Yaskawa INFORM job: R1_W35-36-A2(90,0)KM-OK_MOD.JBI

/JOB
//NAME R1_W35-36-A2(90,0)KM-OK_MOD
///FOLDERNAME KRIS-SCIANA
//POS
///NPOS 134,134,0,9,0,0
///TOOL 0
///POSTYPE PULSE
///PULSE
C00000=-14538,91541,13322,-12188,94395,86333
C00001=-53862,-64636,-102244,-12188,94395,-55972
C00002=-133203,-148839,-120155,9781,61912,-66404
C00003=-174797,-117438,-114286,21839,44085,-72130
C00004=-167772,-84651,-94857,14466,47220,-68129
C00005=-165686,-79015,-89435,12794,46452,-67294
C00006=-164380,-75470,-85062,11842,45407,-66832
C00007=-163956,-74163,-84447,11412,45634,-66605
C00008=-164380,-75470,-85062,11842,45407,-66832
C00009=-164380,-75556,-84437,11929,44986,-66887
C00010=-164380,-75470,-85062,11842,45407,-66832
C00011=-153920,-88332,-89590,-12436,38200,-57880
C00012=-154679,-95973,-95556,-11711,37839,-58237
C00013=-173550,-85808,-91859,28172,44692,-80325
C00014=-171230,-80345,-86542,26466,43532,-79492
C00015=-169766,-76768,-82629,25474,42568,-79023
C00016=-169296,-75560,-82068,24939,42679,-78740
C00017=-169766,-76768,-82629,25474,42568,-79023
C00018=-169766,-76789,-82113,25628,42271,-79117
C00019=-169766,-76768,-82629,25474,42568,-79023
C00020=-181492,-65923,-79959,40723,57193,-83283
C00021=-194013,-96598,-96464,48452,59531,-88352
C00022=-194013,-96598,-96464,48452,59531,50649
C00023=-203995,-41983,-97549,32423,85878,60714
C00024=-215531,-16643,-75179,16986,87607,63817
C00025=-220381,20760,-46740,28196,103428,68967
C00026=-222470,47333,-20175,33789,109715,69761
C00027=-222470,47333,-20175,33789,109715,69761
C00028=-227285,124532,76693,31976,94430,63431
C00029=-227285,124532,76693,347,94430,63431
C00030=-219016,126985,91892,33963,94141,66872
C00031=-220579,120356,82895,34199,96539,66979
C00032=-220443,116751,78046,34294,97429,67310
C00033=-220485,117945,78617,34323,97664,67366
C00034=-220116,109570,67451,34578,99656,68141
C00035=-220116,109383,68055,34523,99266,68019
C00036=-220116,109727,67000,34621,99953,68237
C00037=-220113,113043,61938,35326,103938,69532
C00038=-235601,86931,27868,38520,116104,67576
C00039=-221806,39036,-18377,32558,104968,68512
C00040=-221724,38193,-19154,32548,104980,68545
C00041=-221793,39711,-18991,32681,105579,68702
C00042=-221571,37477,-21115,32657,105643,68801
C00043=-221571,37188,-20943,32612,105427,68735
C00044=-222926,39369,-21029,33153,106861,68698
C00045=-223966,38557,-20553,33262,106600,68250
C00046=-226583,52363,-1545,40953,111419,72507
C00047=-222365,54755,1299,40199,109281,73389
C00048=-223739,53056,-5101,41284,112199,74042
C00049=-218620,25381,-36348,28708,102369,69449
C00050=-215610,6815,-53590,21086,94935,66327
C00051=-215610,6815,-53590,21086,94935,66327
C00052=-181695,43526,-29600,12157,122514,78492
C00053=-175710,40538,-26347,11007,118384,79933
C00054=-175710,39274,-25893,10901,117472,79840
C00055=-175710,38697,-25667,10854,117045,79797
C00056=-175710,39140,-25841,10891,117374,79830
C00057=-179718,48062,-16175,11178,116478,78456
C00058=-179718,47173,-15797,11104,115801,78387
C00059=-179840,45925,-17165,11141,116013,78370
C00060=-180929,50093,-14822,11330,116824,78102
C00061=-186701,42472,-23184,12056,118705,76442
C00062=-186701,42137,-23058,12024,118461,76415
C00063=-186701,41522,-22818,11965,118005,76364
C00064=-186701,41854,-22950,11997,118252,76391
C00065=-186455,49519,-14567,11826,117028,76335
C00066=-186455,48820,-14270,11763,116497,76277
C00067=-186489,47678,-15355,11775,116580,76274
C00068=-186464,50343,-14383,11863,117331,76364
C00069=-197498,47452,-17867,12899,119348,72986
C00070=-197498,47072,-17722,12859,119070,72952
C00071=-197498,46496,-17490,12799,118641,72900
C00072=-197498,47063,-17718,12858,119062,72951
C00073=-196870,55601,-8139,12610,117509,72975
C00074=-196870,54375,-7597,12489,116567,72866
C00075=-196979,52904,-9261,12531,116843,72862
C00076=-197536,57261,-7580,12726,118092,72824
C00077=-207821,57139,-7720,13405,119482,69564
C00078=-207821,56572,-7499,13343,119066,69511
C00079=-207821,55859,-7201,13265,118530,69444
C00080=-207821,56362,-7414,13320,118909,69491
C00081=-206745,64730,2328,13030,117110,69632
C00082=-206745,63773,2776,12932,116361,69543
C00083=-206913,62534,1322,12975,116636,69520
C00084=-207056,64481,1794,13074,117348,69557
C00085=-206807,74763,-1333,14129,124086,70525
C00086=-222470,47333,-20175,33789,109715,69761
C00087=-227285,124532,76693,31976,94430,63431
C00088=-227285,124532,76693,347,94430,63431
C00089=-219683,125196,85472,34228,96937,67464
C00090=-210093,88761,31172,12143,100206,68021
C00091=-211457,88325,33046,12355,99045,67470
C00092=-210790,76646,19815,10799,97227,55457
C00093=-211035,76565,20978,10838,96514,55320
C00094=-215754,68895,15354,21936,91924,55428
C00095=-212561,72725,19936,20957,90379,56197
C00096=-220321,59927,15297,39942,81300,54728
C00097=-221083,58673,11708,40099,82839,55002
C00098=-221083,64899,6113,39881,87997,56947
C00099=-237363,57466,-2523,45822,95924,53882
C00100=-178606,-9643,-70218,5498,91826,76131
C00101=-178606,-14634,-67984,5486,87904,75961
C00102=-178606,-16618,-66817,5490,86174,75885
C00103=-164717,-14931,-65520,-673,85890,79822
C00104=-168728,-34051,-72545,6771,71301,79816
C00105=-174833,-47628,-86367,10104,73375,78049
C00106=-186297,-13357,-69402,-4449,89057,68000
C00107=-188919,-11221,-65810,-3280,87847,67318
C00108=-188919,-13641,-64406,-3283,85743,67372
C00109=-208365,-934,-54515,5411,86403,61879
C00110=-208466,2490,-56744,5454,89524,61986
C00111=-165581,-9313,-66363,-13501,91122,73549
C00112=-173591,2305,-58786,-1879,99187,73604
C00113=-173591,336,-57916,-1870,97641,73627
C00114=-194419,4863,-54227,5414,98069,67881
C00115=-194382,10167,-56400,5486,102112,68070
C00116=-175852,-53507,-90925,10675,73277,77722
C00117=-192163,-97364,-101667,47222,60310,-87268
C00118=-152921,-121523,-105240,-887,29191,-65898
C00119=-145454,-97388,-91369,-9797,33546,-61459
C00120=-145164,-93769,-89182,-10007,34090,-61358
C00121=-145492,-97327,-90174,-9935,32848,-61383
C00122=-144929,-94616,-90367,-10204,34407,-61264
C00123=-144481,-92111,-90249,-8813,37568,-61280
C00124=-144474,-92075,-90268,-8813,37601,-61278
C00125=-146631,-92505,-88658,-8221,34248,-62254
C00126=-145432,-97308,-91545,-9785,33697,-61466
C00127=-146808,-105152,-97390,-8250,33115,-62229
C00128=-157428,-155890,-120182,7201,20895,-69928
C00129=-121608,-155890,-113294,7201,20895,-69928
C00130=-121608,-155890,-113294,7201,20895,-69928
C00131=-6794,-155890,-113294,7201,20895,-69928
C00132=19798,28184,-21106,-6770,70886,39620
C00133=31261,107535,18634,-12792,92436,86844
BC00000=215919,10610,1075157
BC00001=365971,10610,1075157
BC00002=337157,3769,1075169
BC00003=321343,15,1075175
BC00004=321343,15,1075175
BC00005=321343,15,1075175
BC00006=321343,15,1075175
BC00007=321343,15,1075175
BC00008=321343,15,1075175
BC00009=321343,15,1075175
BC00010=321343,15,1075175
BC00011=321343,15,1075175
BC00012=321343,15,1075175
BC00013=358709,15,1075175
BC00014=358709,15,1075175
BC00015=358709,15,1075175
BC00016=358709,15,1075175
BC00017=358709,15,1075175
BC00018=358709,15,1075175
BC00019=358709,15,1075175
BC00020=358709,15,1075175
BC00021=358709,15,1075175
BC00022=358709,15,1075175
BC00023=358709,15,1075175
BC00024=358709,15,1075175
BC00025=358709,15,1075175
BC00026=358709,15,1075175
BC00027=360810,67986,1075175
BC00028=360810,67986,1075175
BC00029=391370,67986,1075175
BC00030=391370,67986,1075175
BC00031=391370,67986,1075175
BC00032=391370,67986,1075175
BC00033=391370,67986,1075175
BC00034=391370,67986,1075175
BC00035=391370,67986,1075175
BC00036=391370,67986,1075175
BC00037=391370,67986,1075175
BC00038=391370,67986,1075175
BC00039=358709,15,1075175
BC00040=358709,15,1075175
BC00041=358709,15,1075175
BC00042=358709,15,1075175
BC00043=358709,15,1075175
BC00044=358709,15,1075175
BC00045=358709,15,1075175
BC00046=358709,15,1075175
BC00047=358709,15,1075175
BC00048=358709,15,1075175
BC00049=358709,15,1075175
BC00050=358709,15,1075175
BC00051=358709,15,1075175
BC00052=358709,15,1075175
BC00053=358709,15,1075175
BC00054=358709,15,1075175
BC00055=358709,15,1075175
BC00056=358709,15,1075175
BC00057=358709,15,1075175
BC00058=358709,15,1075175
BC00059=358709,15,1075175
BC00060=358709,15,1075175
BC00061=358709,15,1075175
BC00062=358709,15,1075175
BC00063=358709,15,1075175
BC00064=358709,15,1075175
BC00065=358709,15,1075175
BC00066=358709,15,1075175
BC00067=358709,15,1075175
BC00068=358709,15,1075175
BC00069=358709,15,1075175
BC00070=358709,15,1075175
BC00071=358709,15,1075175
BC00072=358709,15,1075175
BC00073=358709,15,1075175
BC00074=358709,15,1075175
BC00075=358709,15,1075175
BC00076=358709,15,1075175
BC00077=358709,15,1075175
BC00078=358709,15,1075175
BC00079=358709,15,1075175
BC00080=358709,15,1075175
BC00081=358709,15,1075175
BC00082=358709,15,1075175
BC00083=358709,15,1075175
BC00084=358709,15,1075175
BC00085=358709,15,1075175
BC00086=360810,67986,1075175
BC00087=360810,67986,1075175
BC00088=391370,67986,1075175
BC00089=391370,67986,1075175
BC00090=391370,67986,1075175
BC00091=391370,67986,1075175
BC00092=391370,67986,1075175
BC00093=391370,67986,1075175
BC00094=391370,67986,1075175
BC00095=391370,67986,1075175
BC00096=391370,67986,1075175
BC00097=391370,67986,1075175
BC00098=391370,67986,1075175
BC00099=391370,67986,1075175
BC00100=358709,15,1075175
BC00101=358709,15,1075175
BC00102=358709,15,1075175
BC00103=358709,15,1075175
BC00104=358709,15,1075175
BC00105=358709,15,1075175
BC00106=358709,15,1075175
BC00107=358709,15,1075175
BC00108=358709,15,1075175
BC00109=358709,15,1075175
BC00110=358709,15,1075175
BC00111=358709,15,1075175
BC00112=358709,15,1075175
BC00113=358709,15,1075175
BC00114=358709,15,1075175
BC00115=358709,15,1075175
BC00116=358709,15,1075175
BC00117=358709,15,1075175
BC00118=339950,15,1075175
BC00119=339226,15,1075175
BC00120=338936,15,1075175
BC00121=338936,15,1075175
BC00122=338936,15,1075175
BC00123=304524,15,1075175
BC00124=301197,15,1075175
BC00125=289564,15,1075175
BC00126=289854,15,1075175
BC00127=290578,15,1075175
BC00128=290578,15,1075175
BC00129=290578,15,1075175
BC00130=386899,15,1075175
BC00131=386899,15,1075175
BC00132=204073,419,1075162
BC00133=125260,593,1075157
///POSTYPE BASE
///RECTAN
///RCONF 0,0,0,0,1,0,0,0,0,0,0,0,0,0,0,0,0,0,0,0,0,0,0,0
P00006=2.006,1.622,-0.565,0.0000,0.0000,0.0000
P00021=0.073,2.058,-0.109,0.0000,0.0000,0.0000
P00022=2.006,1.622,-0.565,0.0000,0.0000,0.0000
///RCONF 0,0,0,0,0,0,0,0,0,0,0,0,0,0,0,0,0,0,0,0,0,0,0,0
P00025=3.643,0.007,-2.585,0.0000,0.0000,0.0000
P00030=-0.014,-0.768,0.131,0.0000,0.0000,0.0000
P00031=-0.170,0.039,-0.647,0.0000,0.0000,0.0000
P00032=-0.423,0.157,3.222,0.0000,0.0000,0.0000
P00033=0.854,-1.099,3.047,0.0000,0.0000,0.0000
P00040=2.716,-0.016,3.014,0.0000,0.0000,0.0000
//INST
///DATE 2025/01/20 13:19
///ATTR SC,RW
///GROUP1 RB1,BS1
NOP
'r1_W35-36-A2(90,0)
'Path S1033 (for W914)
SFTOF
MOVJ C00000 BC00000 VJ=20.00
MOVJ C00001 BC00001 VJ=20.00
MOVJ C00002 BC00002 VJ=20.00
MOVJ C00003 BC00003 VJ=20.00
MOVL C00004 BC00004 V=166.7
MOVL C00005 BC00005 V=166.7
MOVL C00006 BC00006 V=60.0
REFP 3 C00007 BC00007
CALL JOB:SEARCH-R1
SET P021 P006
SFTON P021
MOVL C00008 BC00008 V=60.0
REFP 3 C00009 BC00009
CALL JOB:SEARCH-R1
SET P021 P006
SFTON P021
MOVL C00010 BC00010 V=60.0
MOVL C00011 BC00011 V=166.7
MOVL C00012 BC00012 V=166.7
'Path S1034 (for W914)
SFTOF
MOVL C00013 BC00013 V=166.7
MOVL C00014 BC00014 V=166.7
MOVL C00015 BC00015 V=60.0
REFP 3 C00016 BC00016
CALL JOB:SEARCH-R1
SET P022 P006
SFTON P022
MOVL C00017 BC00017 V=60.0
REFP 3 C00018 BC00018
CALL JOB:SEARCH-R1
SET P022 P006
SFTON P022
MOVL C00019 BC00019 V=60.0
MOVL C00020 BC00020 V=166.7
MOVJ C00021 BC00021 VJ=20.00
MOVJ C00022 BC00022 VJ=100.00
MOVJ C00023 BC00023 VJ=100.00
SFTOF
MOVJ C00024 BC00024 VJ=100.00
MOVJ C00025 BC00025 VJ=50.00
MOVJ C00026 BC00026 VJ=60.00
MOVL C00027 BC00027 V=1000.0
MOVL C00028 BC00028 V=1000.0
MOVL C00029 BC00029 V=1000.0
MOVL C00030 BC00030 V=1000.0
MOVL C00031 BC00031 V=166.7
REFP 3 C00032 BC00032
CALL JOB:SEARCH-R1
SET P040 P006
SFTON P040
MOVL C00033 BC00033 V=166.7
MOVL C00034 BC00034 V=166.7
REFP 3 C00035 BC00035
CALL JOB:SEARCH-R1
SET P040 P006
SFTON P040
MOVL C00036 BC00036 V=166.7
SFTOF
MOVL C00037 BC00037 V=666.7
MOVL C00038 BC00038 V=666.7
COMM PAUSE
COMM MOVL C00039 BC00039 V=60.0
COMM REFP 3 C00040 BC00040
COMM CALL JOB:SEARCH-R1
COMM SET P025 P006
COMM SFTON P025
COMM MOVL C00041 BC00041 V=83.3
COMM MOVL C00042 BC00042 V=60.0
COMM REFP 3 C00043 BC00043
COMM CALL JOB:SEARCH-R1
COMM SET P025 P006
COMM SFTON P025
COMM MOVL C00044 BC00044 V=60.0
COMM MOVL C00045 BC00045 V=166.7
COMM MACRO1 MJ#(0) ARGF6
COMM SFTON P025
COMM MOVJ C00046 BC00046 VJ=10.00
COMM MOVL C00047 BC00047 V=13.3
COMM ARCOF
COMM MOVL C00048 BC00048 V=83.3
COMM SFTOF
COMM PAUSE
MOVL C00049 BC00049 V=166.7
MOVJ C00050 BC00050 VJ=20.00
MOVL C00051 BC00051 V=166.7
MOVJ C00052 BC00052 VJ=20.00
MOVL C00053 BC00053 V=233.3
MOVL C00054 BC00054 V=60.0
REFP 3 C00055 BC00055
CALL JOB:SEARCH-R1
SET P030 P006
SFTON P030
MOVL C00056 BC00056 V=60.0
MOVL C00057 BC00057 V=100.0
MOVL C00058 BC00058 V=60.0
REFP 3 C00059 BC00059
CALL JOB:SEARCH-R1
SET P030 P006
SFTON P030
MOVL C00060 BC00060 V=60.0
SFTOF
MOVL C00061 BC00061 V=233.3
MOVL C00062 BC00062 V=60.0
REFP 3 C00063 BC00063
CALL JOB:SEARCH-R1
SET P031 P006
SFTON P031
MOVL C00064 BC00064 V=60.0
MOVL C00065 BC00065 V=100.0
MOVL C00066 BC00066 V=60.0
REFP 3 C00067 BC00067
CALL JOB:SEARCH-R1
SET P031 P006
SFTON P031
MOVL C00068 BC00068 V=60.0
SFTOF
MOVL C00069 BC00069 V=233.3
MOVL C00070 BC00070 V=60.0
REFP 3 C00071 BC00071
CALL JOB:SEARCH-R1
SET P032 P006
SFTON P032
MOVL C00072 BC00072 V=60.0
MOVL C00073 BC00073 V=100.0
MOVL C00074 BC00074 V=60.0
REFP 3 C00075 BC00075
CALL JOB:SEARCH-R1
SET P032 P006
SFTON P032
MOVL C00076 BC00076 V=60.0
SFTOF
MOVL C00077 BC00077 V=233.3
MOVL C00078 BC00078 V=60.0
REFP 3 C00079 BC00079
CALL JOB:SEARCH-R1
SET P033 P006
SFTON P033
MOVL C00080 BC00080 V=60.0
MOVL C00081 BC00081 V=100.0
MOVL C00082 BC00082 V=60.0
REFP 3 C00083 BC00083
CALL JOB:SEARCH-R1
SET P033 P006
SFTON P033
MOVL C00084 BC00084 V=60.0
SFTOF
MOVL C00085 BC00085 V=333.3
MOVL C00086 BC00086 V=1000.0
MOVL C00087 BC00087 V=1000.0
MOVL C00088 BC00088 V=1000.0
MOVL C00089 BC00089 V=1000.0
MOVL C00090 BC00090 V=166.7
CALL JOB:COFNIJ_DRUT
MOVL C00091 BC00091 V=166.7
SFTON P040
MOVL C00092 BC00092 V=166.7
MOVL C00093 BC00093 V=166.7 PL=0
MACRO1 MJ#(0) ARGF7
ARCON
MOVL C00094 BC00094 V=8.3
MOVL C00095 BC00095 V=8.3
MOVL C00096 BC00096 V=8.3
ARCOF
MOVL C00097 BC00097 V=166.7
SFTOF
MOVL C00098 BC00098 V=1000.0
MOVL C00099 BC00099 V=1000.0
MOVL C00100 BC00100 V=333.3
MOVJ C00101 BC00101 VJ=15.00
SFTON P031
MOVL C00102 BC00102 V=100.0 PL=0
MACRO1 MJ#(0) ARGF9
ARCON
SFTON P030
MOVL C00103 BC00103 V=13.3
MOVL C00104 BC00104 V=13.3
ARCOF
MOVL C00105 BC00105 V=166.7
SFTOF
MOVJ C00106 BC00106 VJ=20.00
MOVJ C00107 BC00107 VJ=20.00
SFTON P032
MOVL C00108 BC00108 V=100.0 PL=0
ARCON
SFTON P033
MOVL C00109 BC00109 V=13.3
ARCOF
MOVJ C00110 BC00110 VJ=20.00
SFTOF
MOVJ C00111 BC00111 VJ=50.00
MOVJ C00112 BC00112 VJ=20.00
SFTON P031
MOVL C00113 BC00113 V=100.0 PL=0
ARCON
SFTON P032
MOVL C00114 BC00114 V=13.3
ARCOF
MOVJ C00115 BC00115 VJ=20.00
MOVJ C00116 BC00116 VJ=20.00
MOVJ C00117 BC00117 VJ=50.00
SFTOF
SFTON P022
MOVJ C00118 BC00118 VJ=20.00
MOVJ C00119 BC00119 VJ=20.00
MOVL C00120 BC00120 V=100.0 PL=0
REFP 1 C00121 BC00121
REFP 2 C00122 BC00122
MACRO1 MJ#(0) ARGF7
ARCON
MOVL C00123 BC00123 V=7.5
SFTON P021
MOVL C00124 BC00124 V=7.5
MOVL C00125 BC00125 V=7.5
ARCOF
MOVL C00126 BC00126 V=166.7
MOVL C00127 BC00127 V=166.7
SFTOF
MOVJ C00128 BC00128 VJ=100.00
MOVJ C00129 BC00129 VJ=60.00
MOVJ C00130 BC00130 VJ=100.00
MOVJ C00131 BC00131 VJ=100.00
MOVJ C00132 BC00132 VJ=100.00
MOVJ C00133 BC00133 VJ=100.00
END
